(* IEC 61131-3 sources: lexer_tests/lexers/Structured Text, 3 files *)

(* ---- test.iecst ---- *)
VAR_GLOBAL
    TEST_ARR: ARRAY[0..2] OF WORD;
END_VAR

FUNCTION_BLOCK FB_TEST
    VAR
        iNum: WORD;

    END_VAR
    TEST_ARR[iNum] := 10;
END_FUNCTION_BLOCK

PROGRAM PLC_PRG
    VAR
        iIndex : WORD;
        fbTest: FB_TEST;
    END_VAR
    fbTest(iNum := 0); // Работает
    fbTest(iNum := iIndex); // Не Работает
    TEST_ARR[1] := 10; // Работает
    TEST_ARR[iIndex] := 10; // Не Работает
    D100 := 1;
    TEST_ARR[D100] := 10; // Не Работает

END_PROGRAM

CONST
    MY_TON_D := 2;
    MY_TO_D := 2;
    LIMIT := 7;
END_CONST

ORGANIZATION_BLOCK CYCLE
    (* **********************************************************
    CYCLE - название OB1, он вызывается циклически системой S7.
    Часть 1 : Вызов функционального блока и передача входных величин
    Часть 2 : Чтение выходных величин и вывод с переключением выходов
    ********************************************************** *)
    VAR_TEMP
        systemdata : ARRAY[0..20] OF BYTE; // Область для OB1
    END_VAR
    BEGIN
    (* Part 1 : ************************************************** *)
    ACQUIRE.ACQUIRE_DATA(
        measval_in  := WORD_TO_INT(input),
        newval      := "Input 0.0", // Входной ключ как идентификатор сигнала
        resort      := %PQW10.23,
        funct_sel   := Function_switch,
        newsel      := Coding_switch,
        selection   := Coding
    );

    (* Part 2 : ************************************************* *)
    IF Output_switch THEN // Изменение выхода
        Output := ACQUIRE_DATA.result_out; // Квадратный корень или квадрат
    ELSE
        Output := ACQUIRE_DATA.measval_out; // Измеряемая величина
    END_IF;
END_ORGANIZATION_BLOCK

TYPE Direction (
    DIR_CW, (* по часовой *)
    DIR_CCW  (* против часовой *)
)
END_TYPE

VAR
    xA : BOOL; (* Фаза а *)
    xB : BOOL; (* Фаза б *)
    enDir : Direction; (* Направление движения *)
    udiCount : DINT; (* Счетчик *)
    fbRTA, fbRTB : R_TRIG;
    fbFTA, fbFTB : F_TRIG;
END_VAR

fbRTA(CLK := xA);
fbFTA(CLK := xA);
fbRTB(CLK := xB);
fbFTB(CLK := xB);

IF  (fbRTA.Q AND NOT xB) OR
    (fbFTA.Q AND xB) OR
    (fbRTB.Q AND xA) OR
    (fbFTB.Q AND NOT xA )
THEN
    enDir := Direction.DIR_CW;
    udiCount := udiCount + 1;
ELSE
    enDir := Direction.DIR_CCW;
    udiCount := udiCount - 1;
END_IF;

PROGRAM PLC_PRG
    VAR
        xStart : BOOL := 'dfsfdfd'; // something
        fbTON1 : TON; (*  \. @WE :=  'dfdf' *)
        rValue : REAL; /* Конечное значение */
    END_VAR

    fbTON1(IN := xStart, PT => tDuration);
    IF xStart <> TRUE THEN
    rValue := easeLinear(fbTON1.ET, rFrom, rTo, tDuration);
    END_IF;
    (a = b)ANDc > 10;
    c := (b / 3) * 12**;
    a := CONCAT(a, ':= **'); // a := b
END_PROGRAM

(* ---- SendMessageTIMERS.iecst ---- *)
/* Example on how to send a message/state every x seconds with Structured Text Programming.
 This example uses a state machine logic */

IF MOTOR_ACTIVATED = TRUE THEN

    CASE State OF

        1:
            SendMessage := TRUE;
            State := 2;

        2:
             tonSendMessage(
                IN := ActivateTmr,
                PT := T#3S );

              // (transmitting 1 message every 3 seconds.)
			  // Choose whether to set or clear ActivateTmr

            IF tonSendMessage.Q  THEN
                ActivateTmr := FALSE;
                State := 1;
            ELSE
                 ActivateTmr := TRUE;
            END_IF;
    END_CASE

END_IF

/*  State 2: have to execute the timer with the ActivateTmr set to false to get the reset to take effect.
This is a standard trap for using PLC on delay timers.

Example of setting incorrectly the timer: (transmitting 3 messages per second instead of only 1 every 3 seconds.)

IF MOTOR_ACTIVATED = TRUE THEN

    CASE State OF

        1:
            SendMessage := TRUE;
            State := 2;

        2:
                ActivateTmr := TRUE;

                tonSendMessage(
                IN := ActivateTmr,
                PT := T#3S );

             IF tonSendMessage.Q  THEN

                 ActivateTmr := FALSE;
                State := 1;
    END_CASE

END_IF */

(* ---- state_engine.st ---- *)
//------------------------------------------------------------------------------
//
//  State engine
//
//------------------------------------------------------------------------------

IF STATE = eFaulted THEN

    IF SEV2 OR SEV3                                 THEN STATE := eRoomFaulted;

    ELSIF      RESET_req

       AND NOT (SEV2 OR SEV3)                         THEN STATE := eInit;

    END_IF

ELSIF STATE = eInit THEN

    IF      STARTED_on                              THEN STATE := ePreVent;

    END_IF

ELSIF STATE = ePreVent THEN

    IF      tonPreVent.Q                            THEN STATE := ePreTest;

    END_IF

ELSIF STATE = ePreTest THEN //CHECK TEST COMPLETE

    IF       TestComplete                           THEN STATE := eBleedDown;

    END_IF

ELSIF STATE = eBleedDown THEN //CHECK VXX<VBUS

    IF       Vxx < Vbus                             THEN STATE := ePreStandby;

    END_IF

ELSIF STATE = ePreStandby THEN

    IF     stS1.RUN_on

        OR stS2.RUN_on

        OR stS3.RUN_on                              THEN STATE := ePreStartPurge;

    END_IF

ELSIF STATE = ePreStartPurge THEN

    IF       tonPreStartPurge.Q                     THEN STATE := eStandBy;

    END_IF

ELSIF STATE = eStandby THEN

    IF     stS1.STATE = eStarting

        OR stS2.STATE = eStarting

        OR stS3.STATE = eStarting                   THEN STATE := eStarting;

    END_IF

ELSIF STATE = eStarting THEN

    IF     stS1.STATE = eRunning

        OR stS2.STATE = eRunning

        OR stS3.STATE = eRunning                    THEN STATE := eRunning;

    END_IF

END_IF;

// ------------- Starting/Running to ShuttingDown ---------------------------------

IF STATE = eStarting or STATE = eRunning THEN

    IF   NOT ((stS1.STATE = eStarting)    OR (stS1.STATE = eRunning))

        AND NOT ((stS2.STATE = eStarting) OR (stS2.STATE = eRunning))

        AND NOT ((stS3.STATE = eStarting) OR (stS3.STATE = eRunning))                    THEN STATE := eShuttingDown;

    END_IF

END_IF

// ------------- ShuttingDown to Standby ------------------------------------------

IF STATE = eShuttingDown THEN

    IF     stS1.STATE <= eStandby

       AND stS2.STATE <= eStandby

       AND stS3.STATE <= eStandby                  THEN STATE := eFaulted;

    END_IF

 END_IF

// ------------- Standby and lower to Faulted/Init --------------------------------

IF STATE <= eStandby THEN

    IF SEV2 OR SEV3                                 THEN STATE := eFaulted;

    ELSIF NOT STARTED_on

          AND NOT SEV2

          AND NOT SEV3                              THEN STATE := eInit;

    END_IF

 END_IF
